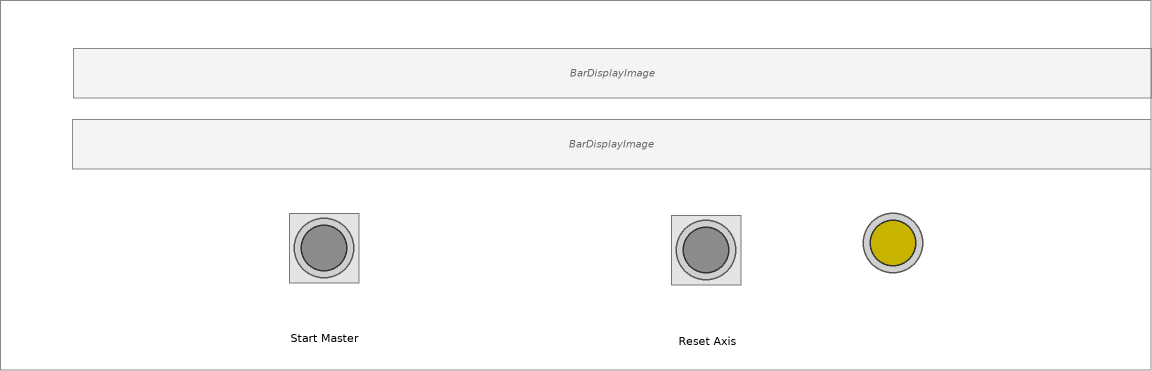
VISUALIZATION Visualization  // 1152x371
    PushSwitch (289,213 70x70), variable: FlyingSaw.bMove, behaviour: TAP, style: Switch-PushSwitch-Gray
    PushSwitch (671,215 70x70), variable: FlyingSaw.bReset, behaviour: TAP, style: Switch-PushSwitch-Gray
    Lamp1 (858,208 70x70), variable: FlyingSaw.bSensor, style: Lamp-Lamp1-Yellow
    BarDisplayImage (73,48 1079x50), value: FlyingSaw.rMasterPosition, style: BarDisplayImage-Gray, scale format: %.1f, scale 0..1440
    BarDisplayImage (72,119 1079x50), value: FlyingSaw.rSlavePosition, style: BarDisplayImage-Gray, scale format: %.1f, scale 0..1440
    Label (240,309 169x59), "Start Master"
    Label (623,312 169x59), "Reset Axis"
END_VISUALIZATION

(* stored: Version 1.1.0.1, ProductVersion 3.1.4024.12
   Visu Visualization: Id {fe4b3744-e8f6-4791-9f2e-59392f43c881} *)
